FUNCTION_BLOCK FB_XpDisableMover
VAR_IN_OUT
	XpMover							: MC_PlanarMover;
	XpGroup							: MC_PlanarGroup;
END_VAR
VAR_INPUT
	execute							: BOOL;
END_VAR
VAR_OUTPUT
	done							: BOOL;
	busy							: BOOL;
	error							: BOOL;
	aborted							: BOOL;
END_VAR
VAR
	_XpFeedback						: ARRAY [0.._MAX_XPLANAR_FEEDBACK] OF MC_PlanarFeedback;
END_VAR
VAR
	_sequence						: UINT;
	_i								: UINT;
	_countError						: UINT;
END_VAR
VAR CONSTANT
	_MAX_XPLANAR_FEEDBACK			: UINT := 1;
	_MAX_COUNT_ERROR				: UINT := 5;
	
	_INIT							: UINT := 0000;
	_READY							: UINT := 0001;
	_REMOVE_FROM_GROUP				: UINT := 0011;
	_CHECK_REMOVE_FROM_GROUP		: UINT := 0012;
	_DISABLE_MOVER					: UINT := 0013;
	_CHECK_DISABLE_MOVER			: UINT := 0014;
	_DONE							: UINT := 1000;
	_ERROR							: UINT := 2000;
	_ABORTED						: UINT := 3000;
END_VAR

updateXPlanarFB();
CASE _sequence OF
	_INIT:
		_sequence := _READY;
		
	_READY:
		IF execute THEN
			busy := TRUE;
			_sequence := _REMOVE_FROM_GROUP;
		END_IF

	_REMOVE_FROM_GROUP:
		XpMover.RemoveFromGroup(commandFeedback:= _XpFeedback[0]);
		_sequence := _CHECK_REMOVE_FROM_GROUP;
	
	_CHECK_REMOVE_FROM_GROUP:
		IF _XpFeedback[0].Done THEN
			_countError := 0;
			_sequence := _DISABLE_MOVER;
		ELSIF _XpFeedback[0].Error THEN
			_countError := _countError + 1;
			_sequence := _REMOVE_FROM_GROUP;
		END_IF
		IF _countError > _MAX_COUNT_ERROR THEN
			_countError := 0;
			_sequence := _ERROR;
		END_IF
	
	_DISABLE_MOVER:
		XpMover.Disable(commandFeedback:= _XpFeedback[1]);
		_sequence := _CHECK_DISABLE_MOVER;
	
	_CHECK_DISABLE_MOVER:
		IF _XpFeedback[1].Done THEN
			_countError := 0;
			_sequence := _DONE;
		ELSIF _XpFeedback[1].Error THEN
			_countError := _countError + 1;
			_sequence := _DISABLE_MOVER;
		END_IF
		IF _countError > _MAX_COUNT_ERROR THEN
			_countError := 0;
			_sequence := _ERROR;
		END_IF
	
	_DONE:
		done := TRUE;
		busy := FALSE;
		IF NOT execute THEN
			done := FALSE;
			_sequence := _READY;
		END_IF
		
	_ERROR:
		error := TRUE;
		busy := FALSE;
		IF NOT execute THEN
			error := FALSE;
			_sequence := _READY;
		END_IF
		
	_ABORTED:
		aborted := TRUE;
		busy := FALSE;
		IF NOT execute THEN
			aborted := FALSE;
			_sequence := _READY;
		END_IF
END_CASE

ACTION updateXPlanarFB:
FOR _i:=0 TO _MAX_XPLANAR_FEEDBACK DO
	_XpFeedback[_i].Update();
END_FOR
END_ACTION

END_FUNCTION_BLOCK

(* stored: Version 1.1.0.1
   POU FB_XpDisableMover: Id {de588409-fa5f-4283-ac2f-376156775266}, SpecialFunc None
   Action updateXPlanarFB: Id {f9db35e4-9497-46d7-9583-edac6b4c33a1} *)
